// Mitsubishi GX Works2 project: 버튼 한 번에 한 동작만 하기   PLC: Q03UDV

PROGRAM MAIN
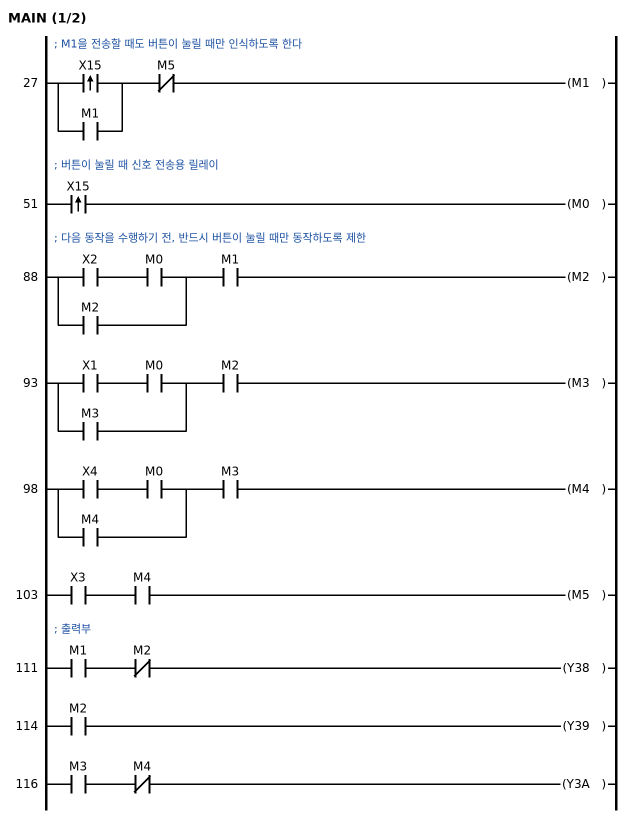
; M1을 전송할 때도 버튼이 눌릴 때만 인식하도록 한다
27    LDP     X15
      OR      M1
      ANI     M5
      OUT     M1
; 버튼이 눌릴 때 신호 전송용 릴레이
51    LDP     X15
      OUT     M0
; 다음 동작을 수행하기 전, 반드시 버튼이 눌릴 때만 동작하도록 제한
88    LD      X2
      AND     M0
      OR      M2
      AND     M1
      OUT     M2
93    LD      X1
      AND     M0
      OR      M3
      AND     M2
      OUT     M3
98    LD      X4
      AND     M0
      OR      M4
      AND     M3
      OUT     M4
103   LD      X3
      AND     M4
      OUT     M5
; 출력부
111   LD      M1
      ANI     M2
      OUT     Y38
114   LD      M2
      OUT     Y39
116   LD      M3
      ANI     M4
      OUT     Y3A
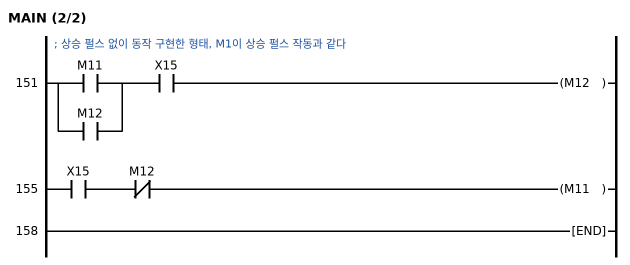
; 상승 펄스 없이 동작 구현한 형태, M1이 상승 펄스 작동과 같다
151   LD      M11
      OR      M12
      AND     X15
      OUT     M12
155   LD      X15
      ANI     M12
      OUT     M11
158   END
END_PROGRAM
